// Mitsubishi GX Works2 project: practice_17   PLC: Q03UDE

PROGRAM MAIN
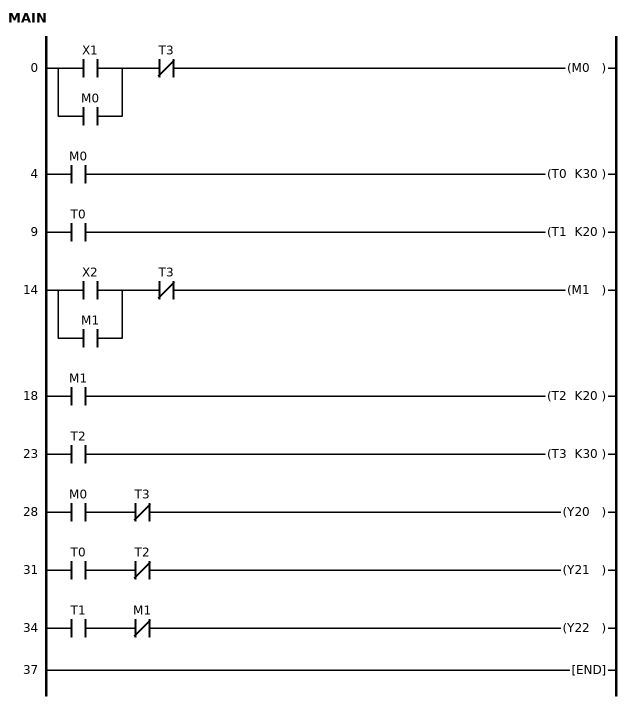
0     LD      X1
      OR      M0
      ANI     T3
      OUT     M0
4     LD      M0
      OUT     T0 K30
9     LD      T0
      OUT     T1 K20
14    LD      X2
      OR      M1
      ANI     T3
      OUT     M1
18    LD      M1
      OUT     T2 K20
23    LD      T2
      OUT     T3 K30
28    LD      M0
      ANI     T3
      OUT     Y20
31    LD      T0
      ANI     T2
      OUT     Y21
34    LD      T1
      ANI     M1
      OUT     Y22
37    END
END_PROGRAM
